(* PLC project actuator, TNI-Software ControlBuild 4.00.17 *)
(* stored: creationDateTime 2005-06-20T11:53:37-01:00 *)

FUNCTION_BLOCK cmd_equipment_library.actuator
  VAR_INPUT  (* CB.group=Modes CB.kind=inputVars *)
    autoMode : BOOL := false;  (* CB.mnemonicPatternPropertyName=<SY>_AUTO_<NU> CB.libelle=Automatic mode *)
    manualMode : BOOL := false;  (* CB.mnemonicPatternPropertyName=<SY>_MANU_<NU> CB.libelle=Manual mode *)
  END_VAR
  VAR_INPUT  (* CB.group=Commands CB.kind=inputVars *)
    autoOpenCmd : BOOL := false;  (* CB.mnemonicPatternPropertyName=<SY>_CMDFWAUTO_<NU> CB.libelle=Automatic open command to the valve *)
    autoCloseCmd : BOOL := false;  (* CB.mnemonicPatternPropertyName=<SY>_CMDSAUTO_<NU> CB.libelle=Automatic close command to the valve *)
  END_VAR
  VAR_INPUT  (* CB.group=PushButtons CB.kind=inputVars *)
    openValvePB : BOOL := false;  (* CB.mnemonicPatternPropertyName=<SY>_BPFW_<NU> CB.libelle=Open valve pushbutton *)
    closeValvePB : BOOL := false;  (* CB.mnemonicPatternPropertyName=<SY>_BPS_<NU> CB.libelle=Close valve pushbutton *)
  END_VAR
  VAR_INPUT  (* CB.group=Sensors CB.kind=inputVars *)
    openedSensorFB : BOOL := false;  (* CB.libelle=Opened sensor feedback *)
    closedSensorFB : BOOL := false;  (* CB.libelle=Closed sensor feedback *)
  END_VAR
  VAR_INPUT  (* CB.kind=inputVars *)
    generalFault : BOOL := false;  (* CB.mnemonicPatternPropertyName=<SY>_DEF_<NU> CB.libelle=General fault of the valve *)
  END_VAR
  VAR_OUTPUT  (* CB.group=Orders CB.kind=outputVars *)
    openCmd : BOOL := false;  (* CB.mnemonicPatternPropertyName=openCmd<SY><NU> CB.libelle=Open command to the valve *)
    closeCmd : BOOL := false;  (* CB.mnemonicPatternPropertyName=closeCmd<SY><NU> CB.libelle=Close command to the valve *)
  END_VAR

(* LD diagram, written out as Structured Text *)
1:
openCmd := (manualMode AND openCmd OR manualMode AND openValvePB AND NOT closeValvePB OR autoMode AND (autoOpenCmd OR openCmd) AND NOT autoCloseCmd) AND NOT openedSensorFB AND NOT generalFault;
2:
closeCmd := (manualMode AND closeCmd OR manualMode AND closeValvePB AND NOT openValvePB OR autoMode AND (autoCloseCmd OR closeCmd) AND NOT autoOpenCmd) AND NOT closedSensorFB AND NOT generalFault;
END_FUNCTION_BLOCK
